{attribute 'qualified_only'}
VAR_GLOBAL
	// Pitch Mechanism:
	{attribute 'TcLinkTo' := '.diEncCnt:=TIIB[EL5042_M1K3_Pitch]^FB Inputs Channel 1^Position'}
	M1K3_Pitch : HOMS_PitchMechanism := (ReqPosLimHi := 1,
		                                 ReqPosLimLo := -1,
		                                 diEncPosLimHi := 1,
		                                 diEncPosLimLo := -1);
END_VAR

(* stored: Version 1.1.0.1, ProductVersion 3.1.4022.18
   GVL GVL_M1K3: Id {c3e91af1-5ac0-497f-aea6-a43e8c284355} *)
